PROGRAM EM01_BoxShorting
VAR
//----Motor-----
	//Barecode Reading	
	FB_BarecodeReadingConv				: MotorManagement;
	stBarecodeReadingConv				: stMotor;
	BarecodeReadingConv_ErrorID			: UINT;
	BarecodeReadingConv_Error			: BOOL;
	bFL_BarecodeReadingConv_Forward		: BOOL;
	//Box Infeed Roller Conveyor 1	
	FB_InfeedRollerConv_1				: MotorManagement;
	stInfeedRollerConv_1				: stMotor;
	InfeedRollerConv_1_ErrorID			: UINT;
	InfeedRollerConv_1_Error			: BOOL;
	bFL_InfeedRollerConv_1_Forward		: BOOL;
	//Box Infeed Roller Conveyor 2	
	FB_InfeedRollerConv_2				: MotorManagement;
	stInfeedRollerConv_2				: stMotor;
	InfeedRollerConv_2_ErrorID			: UINT;
	InfeedRollerConv_2_Error			: BOOL;
	bFL_InfeedRollerConv_2_Forward		: BOOL;
	//Box Infeed Roller Conveyor 3	
	FB_InfeedRollerConv_3				: MotorManagement;
	stInfeedRollerConv_3				: stMotor;
	InfeedRollerConv_3_ErrorID			: UINT;
	InfeedRollerConv_3_Error			: BOOL;
	bFL_InfeedRollerConv_3_Forward		: BOOL;
//----Pneumatic-----
	//Box Pusher for Reject Barcode	
	FB_BoxPusherRejectBarcode			: Pneumatic_1Coil_Management;
	stBoxPusherRejectBarcode			: stPneumatic1;
	BoxPusherRejectBarcode_Error		: BOOL;
	BoxPusherRejectBarcode_ErrorID		: INT;
	BoxPusherRejectBarcode_ErrorMsg		: STRING;
	bFL_BoxPusherRejectBarcode_Adv		: BOOL;
	//Box Pusher for Reject Weight	
	FB_BoxPusherRejectWeight			: Pneumatic_1Coil_Management;
	stBoxPusherRejectWeight				: stPneumatic1;
	BoxPusherRejectWeight_Error			: BOOL;
	BoxPusherRejectWeight_ErrorID		: INT;
	BoxPusherRejectWeight_ErrorMsg		: STRING;
	bFL_BoxPusherRejectWeight_Adv		: BOOL;
	//Box Pusher for Robot	
	FB_BoxPusherRobot					: Pneumatic_1Coil_Management;
	stBoxPusherRobot					: stPneumatic1;
	BoxPusherRobot_Error				: BOOL;
	BoxPusherRobot_ErrorID				: INT;
	BoxPusherRobot_ErrorMsg				: STRING;
	bFL_BoxPusherRobot_Adv				: BOOL;
END_VAR

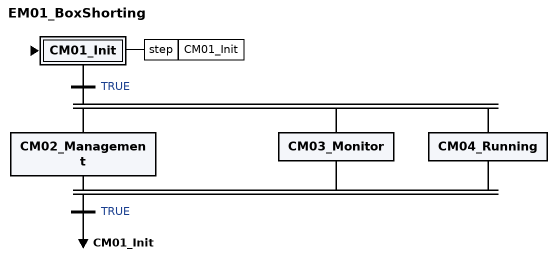
INITIAL_STEP CM01_Init:
    CM01_Init(N);  // step action
END_STEP
TRANSITION FROM CM01_Init TO (CM02_Management, CM03_Monitor, CM04_Running)
    := TRUE;
END_TRANSITION
STEP CM02_Management:
END_STEP
STEP CM03_Monitor:
END_STEP
STEP CM04_Running:
END_STEP
TRANSITION FROM (CM02_Management, CM03_Monitor, CM04_Running) TO CM01_Init
    := TRUE;
END_TRANSITION

ACTION CM01_Init:

END_ACTION

ACTION CM02_Management:
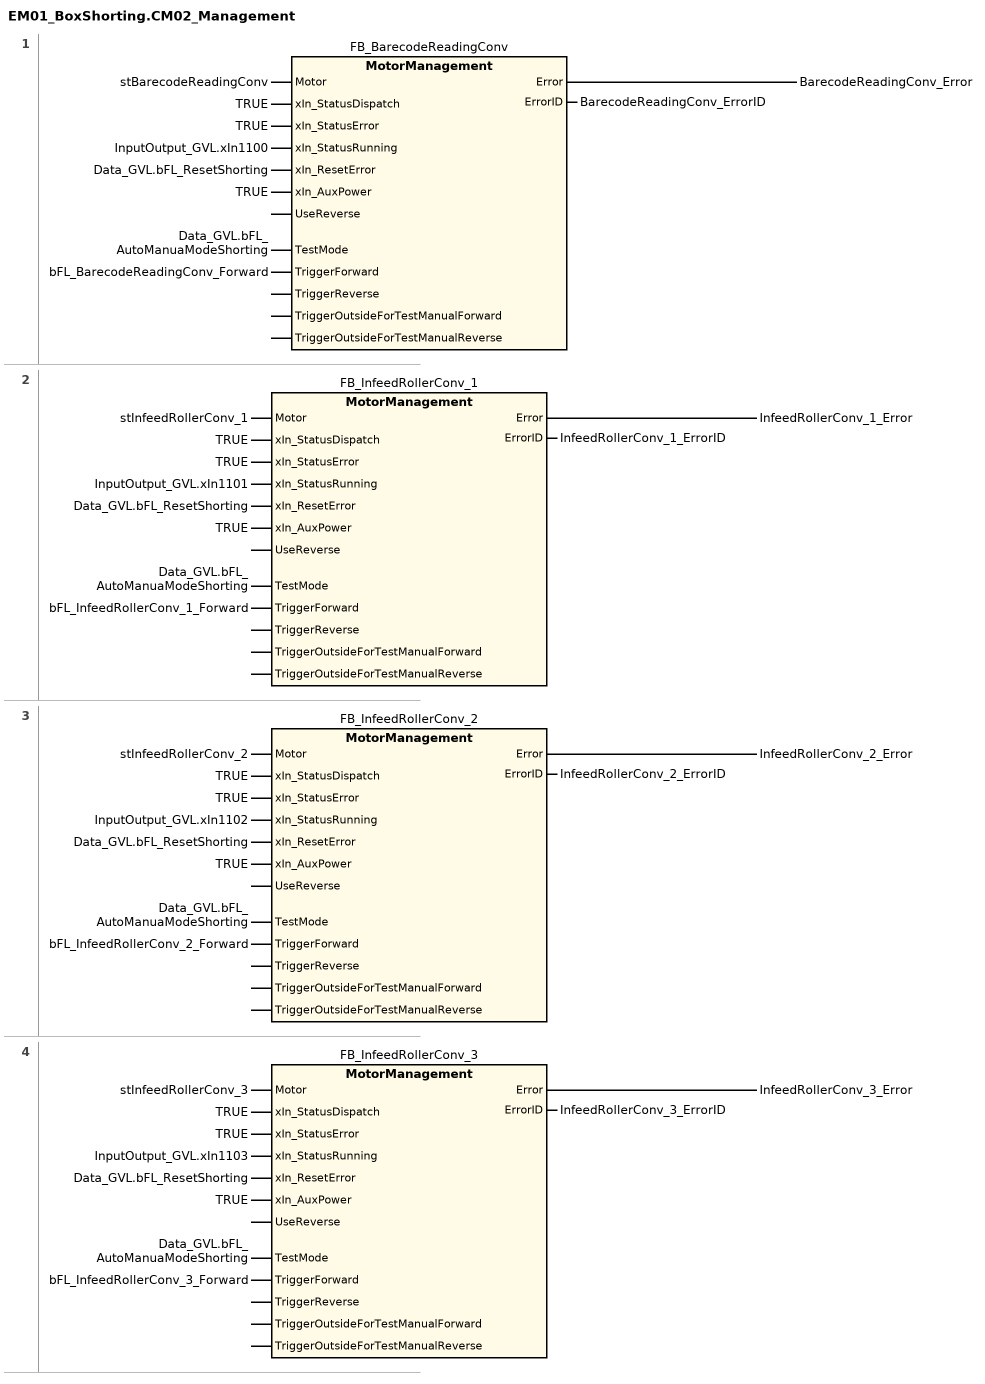
// NETWORK 1
FB_BarecodeReadingConv(
    Motor := stBarecodeReadingConv,
    xIn_StatusDispatch := TRUE,
    xIn_StatusError := TRUE,
    xIn_StatusRunning := InputOutput_GVL.xIn1100,
    xIn_ResetError := Data_GVL.bFL_ResetShorting,
    xIn_AuxPower := TRUE,
    TestMode := Data_GVL.bFL_AutoManuaModeShorting,
    TriggerForward := bFL_BarecodeReadingConv_Forward,
    ErrorID => BarecodeReadingConv_ErrorID); // MotorManagement
BarecodeReadingConv_Error := FB_BarecodeReadingConv.Error;

// NETWORK 2
FB_InfeedRollerConv_1(
    Motor := stInfeedRollerConv_1,
    xIn_StatusDispatch := TRUE,
    xIn_StatusError := TRUE,
    xIn_StatusRunning := InputOutput_GVL.xIn1101,
    xIn_ResetError := Data_GVL.bFL_ResetShorting,
    xIn_AuxPower := TRUE,
    TestMode := Data_GVL.bFL_AutoManuaModeShorting,
    TriggerForward := bFL_InfeedRollerConv_1_Forward,
    ErrorID => InfeedRollerConv_1_ErrorID); // MotorManagement
InfeedRollerConv_1_Error := FB_InfeedRollerConv_1.Error;

// NETWORK 3
FB_InfeedRollerConv_2(
    Motor := stInfeedRollerConv_2,
    xIn_StatusDispatch := TRUE,
    xIn_StatusError := TRUE,
    xIn_StatusRunning := InputOutput_GVL.xIn1102,
    xIn_ResetError := Data_GVL.bFL_ResetShorting,
    xIn_AuxPower := TRUE,
    TestMode := Data_GVL.bFL_AutoManuaModeShorting,
    TriggerForward := bFL_InfeedRollerConv_2_Forward,
    ErrorID => InfeedRollerConv_2_ErrorID); // MotorManagement
InfeedRollerConv_2_Error := FB_InfeedRollerConv_2.Error;

// NETWORK 4
FB_InfeedRollerConv_3(
    Motor := stInfeedRollerConv_3,
    xIn_StatusDispatch := TRUE,
    xIn_StatusError := TRUE,
    xIn_StatusRunning := InputOutput_GVL.xIn1103,
    xIn_ResetError := Data_GVL.bFL_ResetShorting,
    xIn_AuxPower := TRUE,
    TestMode := Data_GVL.bFL_AutoManuaModeShorting,
    TriggerForward := bFL_InfeedRollerConv_3_Forward,
    ErrorID => InfeedRollerConv_3_ErrorID); // MotorManagement
InfeedRollerConv_3_Error := FB_InfeedRollerConv_3.Error;

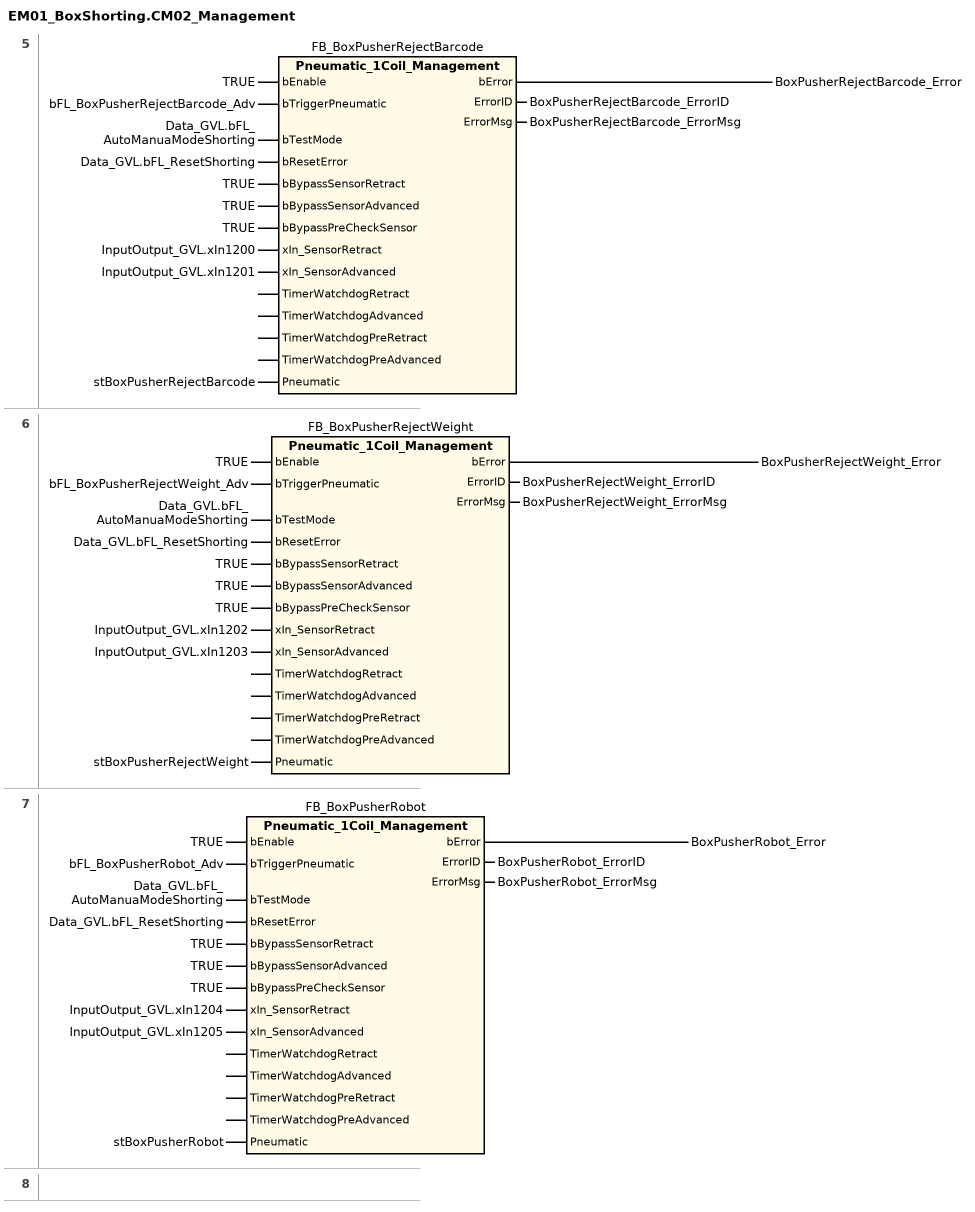
// NETWORK 5
FB_BoxPusherRejectBarcode(
    bEnable := TRUE,
    bTriggerPneumatic := bFL_BoxPusherRejectBarcode_Adv,
    bTestMode := Data_GVL.bFL_AutoManuaModeShorting,
    bResetError := Data_GVL.bFL_ResetShorting,
    bBypassSensorRetract := TRUE,
    bBypassSensorAdvanced := TRUE,
    bBypassPreCheckSensor := TRUE,
    xIn_SensorRetract := InputOutput_GVL.xIn1200,
    xIn_SensorAdvanced := InputOutput_GVL.xIn1201,
    Pneumatic := stBoxPusherRejectBarcode,
    ErrorID => BoxPusherRejectBarcode_ErrorID,
    ErrorMsg => BoxPusherRejectBarcode_ErrorMsg); // Pneumatic_1Coil_Management
BoxPusherRejectBarcode_Error := FB_BoxPusherRejectBarcode.bError;

// NETWORK 6
FB_BoxPusherRejectWeight(
    bEnable := TRUE,
    bTriggerPneumatic := bFL_BoxPusherRejectWeight_Adv,
    bTestMode := Data_GVL.bFL_AutoManuaModeShorting,
    bResetError := Data_GVL.bFL_ResetShorting,
    bBypassSensorRetract := TRUE,
    bBypassSensorAdvanced := TRUE,
    bBypassPreCheckSensor := TRUE,
    xIn_SensorRetract := InputOutput_GVL.xIn1202,
    xIn_SensorAdvanced := InputOutput_GVL.xIn1203,
    Pneumatic := stBoxPusherRejectWeight,
    ErrorID => BoxPusherRejectWeight_ErrorID,
    ErrorMsg => BoxPusherRejectWeight_ErrorMsg); // Pneumatic_1Coil_Management
BoxPusherRejectWeight_Error := FB_BoxPusherRejectWeight.bError;

// NETWORK 7
FB_BoxPusherRobot(
    bEnable := TRUE,
    bTriggerPneumatic := bFL_BoxPusherRobot_Adv,
    bTestMode := Data_GVL.bFL_AutoManuaModeShorting,
    bResetError := Data_GVL.bFL_ResetShorting,
    bBypassSensorRetract := TRUE,
    bBypassSensorAdvanced := TRUE,
    bBypassPreCheckSensor := TRUE,
    xIn_SensorRetract := InputOutput_GVL.xIn1204,
    xIn_SensorAdvanced := InputOutput_GVL.xIn1205,
    Pneumatic := stBoxPusherRobot,
    ErrorID => BoxPusherRobot_ErrorID,
    ErrorMsg => BoxPusherRobot_ErrorMsg); // Pneumatic_1Coil_Management
BoxPusherRobot_Error := FB_BoxPusherRobot.bError;

// NETWORK 8
END_ACTION

ACTION CM03_Monitor:
// NETWORK 1
END_ACTION

ACTION CM04_Running:
// NETWORK 1
END_ACTION

END_PROGRAM

(* stored: Version 1.1.0.1, ProductVersion 3.1.4024.9
   POU EM01_BoxShorting: Id {31edf2cd-c72a-4ec6-9913-4a0997fed385}, SpecialFunc None
   Action CM01_Init: Id {bc17bc7e-7ef1-45a9-85e1-62ec9a9ed2c1}
   Action CM02_Management: Id {b328181f-2066-4349-9588-bb0f5b1345c4}
   Action CM03_Monitor: Id {587ff986-309e-41de-8f65-2cb42ec711ef}
   Action CM04_Running: Id {2acb1116-58e0-4f8b-8bd5-01fe5141f75a} *)
